Yaskawa INFORM job: TEST.JBI

/JOB
//NAME TEST
///FOLDERNAME 03-MASER_SKRZYNIE_TWIN
//POS
///NPOS 0,0,0,0,0,0
//INST
///DATE 2024/10/24 08:33
///ATTR SC,RW,RJ
////FRAME ROBOT
///GROUP1 RB1,BS1
NOP
END
